RoboDK station: RobodkBasico-2.rdk

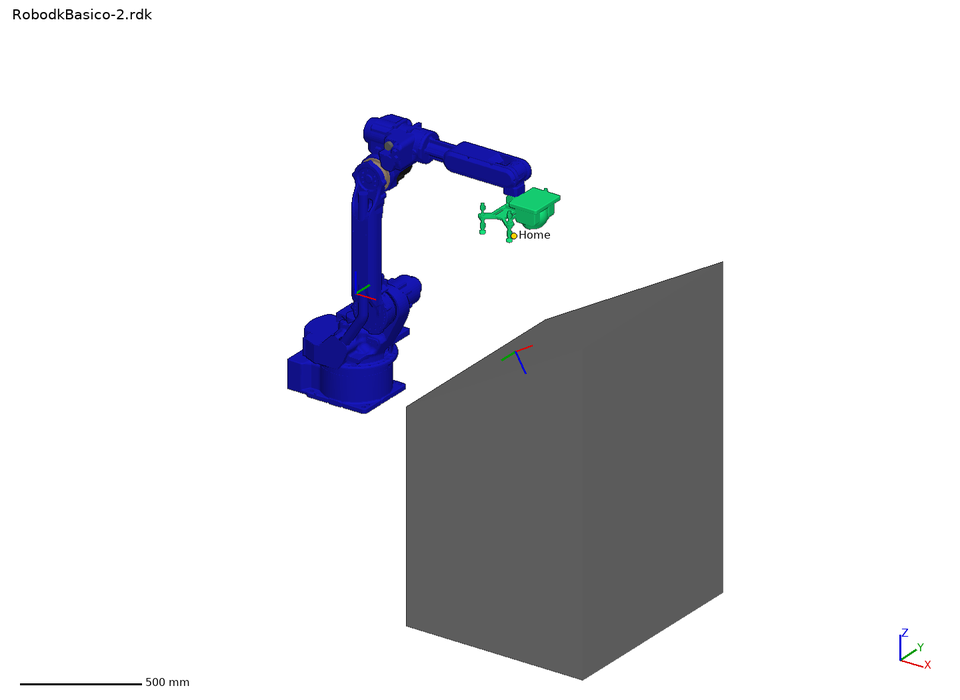
[picture v0: the station drawn from its stored meshes, robots at their saved joint values, targets as dots, program paths as lines]
Station Robodk (2) (saved by RoboDK 5.9.1). Poses are relative to the parent item; angles as X-Y-Z fixed-axis rotations.
  - frame Motoman MH6 Base at (0, 0, 450) mm
    - robot Motoman MH6: 6 axes, payload 6 kg, reach 1422 mm, repeatability 0.08 mm, weight 130 kg
        modified DH rows (alpha deg, a mm, theta deg, d mm): 0, 0, 0, 450; -90, 152, -90, 0; 0, 614, 0, 0; -90, 155, 0, 640; 90, 0, 90, 0; -90, 0, 0, 95
        base shift (0, 0, -450) mm
        joint limits [-170, -90, -175, -180, -45, -360] to [170, 155, 250, 180, 225, 360]; home [0, 0, 0, 0, 0, 0]; saved at [0, 0, 0, 0, 0, 0]
      - tool Ventosas, TCP at (0, 0, 190) mm, size 250 x 290 x 148 mm
    - frame Frame_from_Target1 at (823.2, -34.49, -21.13) mm, rotated rx -180 ry -30 rz 0 deg
      - target Home (Cartesian target) at (225.55, -34.49, -453.06) mm, rotated rx 0 ry -30 rz 0 deg; joints [0, 0, 0, 0, 0, 0] of Motoman MH6
  - object CAJA2 at (1600, 500, 300) mm, rotated rx 180 ry 0 rz 0 deg, size 886.4 x 1000 x 1511.7 mm, geometry from CAJA2.stp
  - Python program RosPolar (listed below)

--- Python program RosPolar ---
from robodk.robolink import *    # API para comunicarte con RoboDK
from robodk.robomath import *    # Funciones matemáticas
import math

#------------------------------------------------
# 1) Conexión a RoboDK e inicialización
#------------------------------------------------
RDK = Robolink()

# Elegir un robot (si hay varios, aparece un popup)
robot = RDK.ItemUserPick("Selecciona un robot", ITEM_TYPE_ROBOT)
if not robot.Valid():
    raise Exception("No se ha seleccionado un robot válido.")

'''
# Conectar al robot físico
if not robot.Connect():
    raise Exception("No se pudo conectar al robot. Verifica que esté en modo remoto y que la configuración sea correcta.")

# Confirmar conexión
if not robot.ConnectedState():
    raise Exception("El robot no está conectado correctamente. Revisa la conexión.")

print("Robot conectado correctamente.")
'''
#------------------------------------------------
# 2) Cargar Frame y Target Home
#------------------------------------------------
frame_name = "Frame_from_Target1"
frame = RDK.Item(frame_name, ITEM_TYPE_FRAME)
if not frame.Valid():
    raise Exception(f'No se encontró el Frame "{frame_name}" en la estación.')

robot.setPoseFrame(frame)
robot.setPoseTool(robot.PoseTool())

# Obtener el Target llamado "Home"
home_target = RDK.Item("Home", ITEM_TYPE_TARGET)
if not home_target.Valid():
    raise Exception('No se encontró un target llamado "Home". Crea uno con ese nombre o cambia el nombre en el código.')

#------------------------------------------------
# 3) Ir a posición Home antes de comenzar
#------------------------------------------------
robot.MoveJ(home_target)

# Ajustes de velocidad y blending
robot.setSpeed(300)   # mm/s
robot.setRounding(5)  # mm

#------------------------------------------------
# 4) Parámetros de la figura (rosa polar)
#------------------------------------------------
num_points = 720
A = 150
n = 5/4  # r = A * sin(n * theta)
z_surface = 0
z_safe = 50

#------------------------------------------------
# 5) Movimiento inicial al centro
#------------------------------------------------
robot.MoveJ(transl(0, 0, z_surface + z_safe))
robot.MoveL(transl(0, 0, z_surface))

#------------------------------------------------
# 6) Dibujar la rosa polar
#------------------------------------------------
turns = 8
max_theta = turns * 2 * math.pi

for i in range(num_points + 1):
    t = i / num_points
    theta = t * max_theta

    r = A * math.sin(n * theta)
    x = r * math.cos(theta)
    y = r * math.sin(theta)

    robot.MoveL(transl(x, y, z_surface))

# Al terminar, subir en Z
robot.MoveL(transl(x, y, z_surface + z_safe))

#------------------------------------------------
# 7) Regresar a Home
#------------------------------------------------
robot.MoveJ(home_target)

print(f"¡Figura completada en el frame '{frame_name}'!")
